INTERFACE I_MachineModule

PROPERTY CfgMachine : REFERENCE TO ST_MachineConfig
GET
END_GET
END_PROPERTY

PROPERTY CmdMachine : REFERENCE TO ST_MachineCommand
GET
END_GET
END_PROPERTY

PROPERTY RcpMachine : REFERENCE TO ST_MachineRecipe
GET
END_GET
END_PROPERTY

PROPERTY StsMachine : REFERENCE TO ST_MachineStatus
GET
END_GET
END_PROPERTY

END_INTERFACE

(* stored: Version 1.1.0.1, ProductVersion 3.1.4024.12
   Itf I_MachineModule: Id {1b8c919d-1463-43ba-aa63-9746ee99167e}
   Property CfgMachine: Id {ac5904f6-49d1-4057-92d2-d0f12b795475}
   Get Get: Id {25a8df1c-ce79-422b-9c49-49b06f5c8b6f}
   Property CmdMachine: Id {ecf12515-bf52-489a-9250-e1618d94752f}
   Get Get: Id {94a361d3-3748-48e1-ad79-5c823cfa3fe4}
   Property RcpMachine: Id {938e5878-6208-4368-8853-13185bfc7d3e}
   Get Get: Id {79134ecd-bd12-4820-9f3a-ff1feeeb6d72}
   Property StsMachine: Id {9ffd5705-26a6-4130-b66c-a5a765360e7e}
   Get Get: Id {bc383727-6ba1-4574-bc40-7ec276904bf7} *)
